INTERFACE ITF

METHOD ITF_METH : STRING
VAR_INPUT
END_VAR
END_METHOD

END_INTERFACE

(* stored: Version 1.1.0.1, ProductVersion 3.1.4022.10
   Itf ITF: Id {75ab29dd-746a-4950-8317-f556b246b006}
   Method ITF_METH: Id {f4394ef9-da8f-4725-9869-01803c1b73ae} *)
